(* CoDeSys 2.3 export: IED_STATE_SYNC.EXP *)

(* POU IED_STATE_SYNC, ST *)
FUNCTION_BLOCK IED_STATE_SYNC
VAR_INPUT
	IED_CONNECT: INT;
END_VAR
VAR_OUTPUT
	IED_STATE: INT;
END_VAR
VAR
END_VAR
IF	IED_CONNECT = 1
	THEN	IED_STATE := 1;
	ELSE	IED_STATE := 0;
END_IF
END_FUNCTION_BLOCK
